(* IEC 61131-3 sources: RL_MAR/experiments/comparison/llm4plc/results/Qwen-Qwen3.5-9B_20260506_150728/20260506_171050, 4 files *)

(* ---- generated_code_iteration_0.st ---- *)
START_ST
FUNCTION_BLOCK TheaterControl
VAR_INPUT
    StartButton : BOOL; (* Input for starting a performance *)
    StopButton : BOOL; (* Input for stopping a performance *)
    SceneNumber : INT; (* Input for selecting the scene or act *)
END_VAR
VAR_OUTPUT
    LightingControl : BOOL; (* Output for controlling lighting *)
    SoundControl : BOOL; (* Output for controlling sound *)
    PerformanceInProgress : BOOL; (* Indicator for an ongoing performance *)
END_VAR
VAR
    state : INT; (* The current FSM state: 0=IDLE, 1=RUNNING, 2=STOPPED *)
    prevStartButton : BOOL; (* Previous state of StartButton for edge detection *)
    prevStopButton : BOOL; (* Previous state of StopButton for edge detection *)
    isValidScene : BOOL; (* Temporary variable to check if SceneNumber is valid *)
END_VAR

BEGIN
    (* --- Step 1: Validate Scene Number --- *)
    (* Check if SceneNumber is 1, 2, or 3 *)
    IF (SceneNumber >= 1) AND (SceneNumber <= 3) THEN
        isValidScene := TRUE;
    ELSE
        isValidScene := FALSE;
    END_IF;

    (* --- Step 2: State Machine Logic --- *)

    (* Transition Logic: Determine Next State *)
    (*
       State 0 (IDLE) -> State 1 (RUNNING):
       Condition: StartButton is TRUE (Rising Edge) AND StopButton is FALSE AND isValidScene is TRUE.
       Note: We use rising edge detection (StartButton AND NOT prevStartButton) to ensure
       the performance starts only once per press, preventing toggling if the button is held.
    *)
    (*
       State 1 (RUNNING) -> State 2 (STOPPED):
       Condition: StopButton is TRUE.
    *)
    (*
       State 2 (STOPPED) -> State 0 (IDLE):
       Condition: StopButton is FALSE AND StartButton is FALSE.
       (If StartButton is still TRUE in State 2, it will transition to State 1 in the next cycle,
        effectively allowing immediate restart if the button remains held, which satisfies the
        "override" requirement while allowing intentional restart).
    *)

    (* Calculate Next State based on current inputs and previous state *)
    CASE state OF
        0: (* IDLE *)
            (* Transition to RUNNING if StartButton rises, Stop is false, and scene is valid *)
            IF (StartButton = TRUE) AND (prevStartButton = FALSE) AND (StopButton = FALSE) AND (isValidScene = TRUE) THEN
                state := 1; (* Transition to RUNNING *)
            ELSE
                state := 0; (* Remain in IDLE *)
            END_IF;

        1: (* RUNNING *)
            (* Transition to STOPPED if StopButton is pressed *)
            IF StopButton = TRUE THEN
                state := 2; (* Transition to STOPPED *)
            ELSE
                state := 1; (* Remain in RUNNING *)
            END_IF;

        2: (* STOPPED *)
            (* Transition to IDLE if StopButton is released and StartButton is not held *)
            (* If StartButton is held while Stop is released, it transitions to RUNNING immediately *)
            IF (StopButton = FALSE) AND (StartButton = FALSE) THEN
                state := 0; (* Transition to IDLE *)
            ELSE
                state := 2; (* Remain in STOPPED until conditions change *)
            END_IF;
    ENDCASE;

    (* --- Step 3: Update Previous Button States --- *)
    (* Store current button states for the next cycle's edge detection *)
    prevStartButton := StartButton;
    prevStopButton := StopButton;

    (* --- Step 4: Assign Outputs Based on Current State --- *)
    CASE state OF
        0: (* IDLE *)
            LightingControl := FALSE;
            SoundControl := FALSE;
            PerformanceInProgress := FALSE;

        1: (* RUNNING *)
            (* Outputs are driven by the validity of the scene number *)
            IF isValidScene = TRUE THEN
                LightingControl := TRUE;
                SoundControl := TRUE;
                PerformanceInProgress := TRUE;
            ELSE
                (* If an invalid scene was selected while trying to start,
                   the state machine logic above prevents entering state 1,
                   but as a safety fallback or if logic changes, ensure outputs are off *)
                LightingControl := FALSE;
                SoundControl := FALSE;
                PerformanceInProgress := FALSE;
            END_IF;

        2: (* STOPPED *)
            LightingControl := FALSE;
            SoundControl := FALSE;
            PerformanceInProgress := FALSE;
    ENDCASE;

END_FUNCTION_BLOCK
END_ST

(* ---- generated_code_iteration_2.st ---- *)
START_REASON
The previous code failed with the error "未知的类型: 'T_TheaterState'" (Unknown type: 'T_TheaterState').

**Root Cause Analysis:**
In IEC 61131-3 Structured Text, `TYPE` definitions must be placed in the **global scope** (outside of any function, function block, or program) to be accessible by other blocks. The previous code attempted to define the `TYPE` inside the `FUNCTION_BLOCK` body, which is syntactically invalid. The compiler could not resolve the type `T_TheaterState` because it was declared locally where it was not allowed.

**Fix Strategy:**
1.  Move the `TYPE T_TheaterState` definition to the global scope, before the `FUNCTION_BLOCK` declaration.
2.  Ensure the `FUNCTION_BLOCK` uses the global type correctly.
3.  Maintain the `FUNCTION_BLOCK` structure and `END_VAR` usage as required.
END_REASON

START_ST
TYPE T_TheaterState :
    IDLE := 0,
    RUNNING := 1,
    STOPPED := 2
END_TYPE;

FUNCTION_BLOCK TheaterControl
VAR_INPUT
    StartButton : BOOL;
    StopButton : BOOL;
    SceneNumber : INT;
END_VAR
VAR_OUTPUT
    LightingControl : BOOL;
    SoundControl : BOOL;
    PerformanceInProgress : BOOL;
END_VAR
VAR
    state : T_TheaterState;
    prevStartButton : BOOL;
    prevStopButton : BOOL;
    isValidScene : BOOL;
END_VAR

BEGIN
    (* --- Step 1: Validate Scene Number --- *)
    IF (SceneNumber >= 1) AND (SceneNumber <= 3) THEN
        isValidScene := TRUE;
    ELSE
        isValidScene := FALSE;
    END_IF;

    (* --- Step 2: State Machine Logic --- *)

    CASE state OF
        IDLE:
            IF (StartButton = TRUE) AND (prevStartButton = FALSE) AND (StopButton = FALSE) AND (isValidScene = TRUE) THEN
                state := RUNNING;
            ELSE
                state := IDLE;
            END_IF;

        RUNNING:
            IF StopButton = TRUE THEN
                state := STOPPED;
            ELSE
                state := RUNNING;
            END_IF;

        STOPPED:
            IF (StopButton = FALSE) AND (StartButton = FALSE) THEN
                state := IDLE;
            ELSE
                state := STOPPED;
            END_IF;
    END_CASE;

    (* --- Step 3: Update Previous Button States --- *)
    prevStartButton := StartButton;
    prevStopButton := StopButton;

    (* --- Step 4: Assign Outputs Based on Current State --- *)
    CASE state OF
        IDLE:
            LightingControl := FALSE;
            SoundControl := FALSE;
            PerformanceInProgress := FALSE;

        RUNNING:
            IF isValidScene = TRUE THEN
                LightingControl := TRUE;
                SoundControl := TRUE;
                PerformanceInProgress := TRUE;
            ELSE
                LightingControl := FALSE;
                SoundControl := FALSE;
                PerformanceInProgress := FALSE;
            END_IF;

        STOPPED:
            LightingControl := FALSE;
            SoundControl := FALSE;
            PerformanceInProgress := FALSE;
    END_CASE;

END_FUNCTION_BLOCK
END_ST

(* ---- generated_code_iteration_3.st ---- *)
START_REASON
The previous code failed due to a character encoding issue. The error message `'gbk' codec can't decode byte 0xaa` indicates that the code contains non-ASCII characters (likely Chinese comments or keywords from a previous attempt or copy-paste error) that are not compatible with the expected ASCII/UTF-8 encoding for the IEC 61131-3 compiler. Specifically, the phrase "未知的类型" (Unknown type) in the previous error log suggests Chinese characters were present in the logic or comments, causing the parser to fail immediately.

To fix this:
1.  Remove all non-ASCII characters (Chinese text) from the code.
2.  Replace them with standard English comments.
3.  Ensure the `TYPE` definition is in the global scope (which was correctly done in the previous iteration, so we keep that structure).
4.  Verify strict adherence to IEC 61131-3 syntax.
END_REASON

START_ST
TYPE T_TheaterState :
    IDLE := 0,
    RUNNING := 1,
    STOPPED := 2
END_TYPE;

FUNCTION_BLOCK TheaterControl
VAR_INPUT
    StartButton : BOOL;
    StopButton : BOOL;
    SceneNumber : INT;
END_VAR
VAR_OUTPUT
    LightingControl : BOOL;
    SoundControl : BOOL;
    PerformanceInProgress : BOOL;
END_VAR
VAR
    state : T_TheaterState;
    prevStartButton : BOOL;
    prevStopButton : BOOL;
    isValidScene : BOOL;
END_VAR

BEGIN
    (* --- Step 1: Validate Scene Number --- *)
    IF (SceneNumber >= 1) AND (SceneNumber <= 3) THEN
        isValidScene := TRUE;
    ELSE
        isValidScene := FALSE;
    END_IF;

    (* --- Step 2: State Machine Logic --- *)

    CASE state OF
        IDLE:
            IF (StartButton = TRUE) AND (prevStartButton = FALSE) AND (StopButton = FALSE) AND (isValidScene = TRUE) THEN
                state := RUNNING;
            ELSE
                state := IDLE;
            END_IF;

        RUNNING:
            IF StopButton = TRUE THEN
                state := STOPPED;
            ELSE
                state := RUNNING;
            END_IF;

        STOPPED:
            IF (StopButton = FALSE) AND (StartButton = FALSE) THEN
                state := IDLE;
            ELSE
                state := STOPPED;
            END_IF;
    END_CASE;

    (* --- Step 3: Update Previous Button States --- *)
    prevStartButton := StartButton;
    prevStopButton := StopButton;

    (* --- Step 4: Assign Outputs Based on Current State --- *)
    CASE state OF
        IDLE:
            LightingControl := FALSE;
            SoundControl := FALSE;
            PerformanceInProgress := FALSE;

        RUNNING:
            IF isValidScene = TRUE THEN
                LightingControl := TRUE;
                SoundControl := TRUE;
                PerformanceInProgress := TRUE;
            ELSE
                LightingControl := FALSE;
                SoundControl := FALSE;
                PerformanceInProgress := FALSE;
            END_IF;

        STOPPED:
            LightingControl := FALSE;
            SoundControl := FALSE;
            PerformanceInProgress := FALSE;
    END_CASE;

END_FUNCTION_BLOCK
END_ST

(* ---- generated_code_iteration_1.st ---- *)
START_REASON
The previous code failed CODESYS compiler validation (Error 500) primarily due to the use of the `CASE` statement with integer literals (`0`, `1`, `2`) as selectors in a `FUNCTION_BLOCK`. While standard IEC 61131-3 allows this, many strict CODESYS compilers (especially older versions or specific configurations) require the `CASE` selector to be of a specific enumerated type or require the `END_CASE` keyword instead of `ENDCASE` if the syntax is slightly off.

However, the most robust fix for CODESYS ST is to:
1.  Define an `ENUM` type for the states to ensure type safety and readability.
2.  Replace the integer literals in the `CASE` statements with the enum values.
3.  Ensure all keywords are spelled correctly (`END_CASE` is the standard, though `ENDCASE` is often accepted, `END_CASE` is safer).
4.  Remove comments that start with `(*` inside the `BEGIN` block if they are causing parsing issues in very strict modes, though usually comments are fine. The main culprit is often the mix of integer literals in CASE without a declared enum type in strict environments.

I will refactor the code to use a dedicated `ENUM` for states and ensure strict compliance with CODESYS syntax.
END_REASON

START_ST
FUNCTION_BLOCK TheaterControl
VAR_INPUT
    StartButton : BOOL;
    StopButton : BOOL;
    SceneNumber : INT;
END_VAR
VAR_OUTPUT
    LightingControl : BOOL;
    SoundControl : BOOL;
    PerformanceInProgress : BOOL;
END_VAR
VAR
    state : T_TheaterState;
    prevStartButton : BOOL;
    prevStopButton : BOOL;
    isValidScene : BOOL;
END_VAR

TYPE T_TheaterState :
    IDLE := 0,
    RUNNING := 1,
    STOPPED := 2
END_TYPE;

BEGIN
    (* --- Step 1: Validate Scene Number --- *)
    IF (SceneNumber >= 1) AND (SceneNumber <= 3) THEN
        isValidScene := TRUE;
    ELSE
        isValidScene := FALSE;
    END_IF;

    (* --- Step 2: State Machine Logic --- *)

    CASE state OF
        IDLE:
            IF (StartButton = TRUE) AND (prevStartButton = FALSE) AND (StopButton = FALSE) AND (isValidScene = TRUE) THEN
                state := RUNNING;
            ELSE
                state := IDLE;
            END_IF;

        RUNNING:
            IF StopButton = TRUE THEN
                state := STOPPED;
            ELSE
                state := RUNNING;
            END_IF;

        STOPPED:
            IF (StopButton = FALSE) AND (StartButton = FALSE) THEN
                state := IDLE;
            ELSE
                state := STOPPED;
            END_IF;
    END_CASE;

    (* --- Step 3: Update Previous Button States --- *)
    prevStartButton := StartButton;
    prevStopButton := StopButton;

    (* --- Step 4: Assign Outputs Based on Current State --- *)
    CASE state OF
        IDLE:
            LightingControl := FALSE;
            SoundControl := FALSE;
            PerformanceInProgress := FALSE;

        RUNNING:
            IF isValidScene = TRUE THEN
                LightingControl := TRUE;
                SoundControl := TRUE;
                PerformanceInProgress := TRUE;
            ELSE
                LightingControl := FALSE;
                SoundControl := FALSE;
                PerformanceInProgress := FALSE;
            END_IF;

        STOPPED:
            LightingControl := FALSE;
            SoundControl := FALSE;
            PerformanceInProgress := FALSE;
    END_CASE;

END_FUNCTION_BLOCK
END_ST
